// TwinCAT 3 PLC project ConvergeStation
// ProgramVersion: 3.1.4026.26
// libraries:
//   Tc2_ModbusRTU, * (Beckhoff Automation GmbH)
//   Tc2_ModbusSrv, * (Beckhoff Automation GmbH)
//   Tc2_Standard, * (Beckhoff Automation GmbH)
//   Tc2_System, * (Beckhoff Automation GmbH)
// project tree:
//   DUTs/ ST_Outputs.TcDUT
//   GVLs/ GVL.TcGVL, IO.TcGVL
//   / PlcTask.TcTTO
//   POUs/Function Blocks/ FB_Intlk.TcPOU, FB_Motors.TcPOU, FB_Sensors.TcPOU
//   POUs/ MAIN.TcPOU
//   POUs/COMM/ FIO_Read_Inputs.TcPOU, FIO_Write_Outputs.TcPOU, ReadWriteIO.TcPOU
//   POUs/PRG/PRG_CTRL/ PRG_CONTROLM1.TcPOU
//   POUs/PRG/ PRG_Mainprg.TcPOU
//   POUs/PRG/PRG_MOTORS/ PRG_Conveyor01.TcPOU, PRG_ExitConvetor.TcPOU, PRG_Load01.TcPOU, PRG_Conveyor02.TcPOU, PRG_Load02.TcPOU, PRG_TransferLeft02.TcPOU, PRG_TransferLeft01.TcPOU
//   POUs/PRG/PRG_SENSORS/ PRG_AtEntry01.TcPOU, PRG_AtExit01.TcPOU, PRG_AtEntry02.TcPOU, PRG_AtTransfer02.TcPOU, PRG_AtTransfer01.TcPOU
// real-time tasks:
//   TASK PlcTask: cycle T#10ms, priority 20, ADS port 350

CONFIGURATION ConvergeStation
    RESOURCE PLC ON TwinCAT3
        TASK PlcTask(INTERVAL := T#10ms, PRIORITY := 20);
        PROGRAM MAIN WITH PlcTask : MAIN;
    END_RESOURCE
END_CONFIGURATION

// ---- DUTs/ST_Outputs.TcDUT
TYPE ST_Outputs :
STRUCT
	Conveyor_1 : BOOL;
	Load_1 : BOOL;
	Unload_1 : BOOL;
	Transfer_Right_1 : BOOL;
	Transfer_Left_1 : BOOL;
	Conveyor_2: BOOL;
	Load_2 : BOOL;
	Unload_2 : BOOL;
	Transfer_Right_2 : BOOL;
	Transfer_Left_2 : BOOL;
	Exit_Conveyor: BOOL;
	Start_Light: BOOL;
	Reset_Light : BOOL;
	Stop_Light: BOOL;
	Counter : INT;
END_STRUCT
END_TYPE

// ---- GVLs/GVL.TcGVL
{attribute 'qualified_only'}
VAR_GLOBAL
	ReadInputs : FB_MBReadInputs;
	WriteCoils : FB_MBWriteCoils;
	FIO_Inputs : ARRAY [0..15] OF BYTE;
	FIO_Outputs : ARRAY [0..15] OF BYTE;
	StartMachine : BOOL;
	Conveyor01OKToRun : BOOL;
	Conveyor02OKToRun : BOOL;
	AtExitPulse : BOOL;
	TransferOKToStart : BOOL;
END_VAR

// ---- GVLs/IO.TcGVL

VAR_GLOBAL
	At_Entry_1 : BOOL;
	At_Entry_2 : BOOL;
	At_Transfer_1 : BOOL;
	At_Transfer_2 : BOOL;
	At_Exit : BOOL;
	Start : BOOL;
	Reset : BOOL;
	Stop : BOOL;
	Emergency_Stop : BOOL;
	Auto : BOOL;
	
	Conveyor_1 : BOOL;
	Load_1 : BOOL;
	Unload_1 : BOOL;
	Transfer_Right_1 : BOOL;
	Transfer_Left_1 : BOOL;
	Conveyor_2 : BOOL;
	Load_2 : BOOL;
	Unload_2 : BOOL;
	Transfer_Right_2 : BOOL;
	Transfer_Left_2 : BOOL;
	Exit_Conveyor : BOOL;
	Start_Light : BOOL;
	Reset_Light : BOOL;
	Stop_Light : BOOL;
END_VAR

// ---- POUs/MAIN.TcPOU
PROGRAM MAIN
VAR
END_VAR

PRG_Mainprg();
PRG_CONTROLM1();

FIO_Read_Inputs();
FIO_Write_Outputs();
ReadWriteIO();

END_PROGRAM

// ---- POUs/PRG/PRG_Mainprg.TcPOU
PROGRAM PRG_Mainprg
VAR
END_VAR

PRG_Conveyor01();
PRG_Conveyor02();
PRG_ExitConvetor();
PRG_Load01();
PRG_Load02();
PRG_TransferLeft01();
PRG_TransferLeft02();

PRG_AtEntry01();
PRG_AtEntry02();
PRG_AtExit01();
PRG_AtTransfer01();
PRG_AtTransfer02();

END_PROGRAM

// ---- POUs/PRG/PRG_MOTORS/PRG_Conveyor01.TcPOU
PROGRAM PRG_Conveyor01
VAR
	intnFBMotor : FB_Motors;
	intnFBIntlk : FB_Intlk;
END_VAR

intnFBIntlk (
	BackwardsInterlock01 := TRUE,
	BackwardsInterlock02 := TRUE,
	BackwardsInterlock03 := TRUE,
	BackwardsInterlock04 := TRUE,
	BackwardsInterlock05 := TRUE,
	ForwardInterlock01 := GVL.Conveyor01OKToRun,
	ForwardInterlock02 := TRUE,
	ForwardInterlock03 := TRUE,
	ForwardInterlock04 := TRUE,
	ForwardInterlock05 := TRUE,
	oStsInterlockOK => intnFBMotor.inIntlkOK,
);

intnFBMotor (
	inStart := GVL.StartMachine,
	outOTE => Conveyor_1,
);

END_PROGRAM

// ---- POUs/Function Blocks/FB_Motors.TcPOU
FUNCTION_BLOCK FB_Motors
VAR_INPUT
	inIntlkOK : BOOL;
	inStart : BOOL;
END_VAR
VAR_OUTPUT
	outOTE: BOOL;
	outRunning : bool;
	outStopped : BOOL;
END_VAR
VAR
END_VAR

IF inIntlkOK AND inStart THEN
	outOTE := TRUE;
	outRunning := TRUE;
	outStopped := FALSE;
	ELSE
	outStopped := TRUE;
	outRunning := FALSE;
	outOTE := FALSE;
END_IF

END_FUNCTION_BLOCK

// ---- POUs/Function Blocks/FB_Intlk.TcPOU
FUNCTION_BLOCK PUBLIC FB_Intlk
VAR_INPUT
	ForwardInterlock01, ForwardInterlock02, ForwardInterlock03, ForwardInterlock04, ForwardInterlock05: BOOL;
	BackwardsInterlock01, BackwardsInterlock02, BackwardsInterlock03, BackwardsInterlock04, BackwardsInterlock05 : BOOL;
END_VAR
VAR_OUTPUT
	oStsInterlockOK : BOOL;
END_VAR
VAR
END_VAR

oStsInterlockOK := 	ForwardInterlock01 AND 
					ForwardInterlock02 AND 
					ForwardInterlock03 AND 
					ForwardInterlock04 AND 
					ForwardInterlock05 AND 
					BackwardsInterlock01 AND 
					BackwardsInterlock02 AND 
					BackwardsInterlock03 AND 
					BackwardsInterlock04 AND 
					BackwardsInterlock05;

END_FUNCTION_BLOCK

// ---- POUs/PRG/PRG_MOTORS/PRG_Conveyor02.TcPOU
PROGRAM PRG_Conveyor02
VAR
	intnFBMotor : FB_Motors;
	intnFBIntlk : FB_Intlk;
END_VAR

intnFBIntlk (
	BackwardsInterlock01 := TRUE,
	BackwardsInterlock02 := TRUE,
	BackwardsInterlock03 := TRUE,
	BackwardsInterlock04 := TRUE,
	BackwardsInterlock05 := TRUE,
	ForwardInterlock01 := GVL.Conveyor02OKToRun,
	ForwardInterlock02 := TRUE,
	ForwardInterlock03 := TRUE,
	ForwardInterlock04 := TRUE,
	ForwardInterlock05 := TRUE,
	oStsInterlockOK => intnFBMotor.inIntlkOK,
);

intnFBMotor (
	inStart := GVL.StartMachine,
	outOTE => Conveyor_2,
);

END_PROGRAM

// ---- POUs/PRG/PRG_MOTORS/PRG_ExitConvetor.TcPOU
PROGRAM PRG_ExitConvetor
VAR
	intnFBMotor : FB_Motors;
	intnFBIntlk : FB_Intlk;
END_VAR

intnFBIntlk (
	BackwardsInterlock01 := TRUE,
	BackwardsInterlock02 := TRUE,
	BackwardsInterlock03 := TRUE,
	BackwardsInterlock04 := TRUE,
	BackwardsInterlock05 := TRUE,
	ForwardInterlock01 := TRUE,
	ForwardInterlock02 := TRUE,
	ForwardInterlock03 := TRUE,
	ForwardInterlock04 := TRUE,
	ForwardInterlock05 := TRUE,
	oStsInterlockOK => intnFBMotor.inIntlkOK,
);

intnFBMotor (
	inStart := GVL.StartMachine,
	outOTE => Exit_Conveyor,
);

END_PROGRAM

// ---- POUs/PRG/PRG_MOTORS/PRG_Load01.TcPOU
PROGRAM PRG_Load01
VAR
	intnFBMotor : FB_Motors;
	intnFBIntlk : FB_Intlk;
END_VAR

intnFBIntlk (
	BackwardsInterlock01 := TRUE,
	BackwardsInterlock02 := TRUE,
	BackwardsInterlock03 := TRUE,
	BackwardsInterlock04 := TRUE,
	BackwardsInterlock05 := TRUE,
	ForwardInterlock01 := NOT PRG_TransferLeft01.intnFBMotor.outRunning,
	ForwardInterlock02 := TRUE,
	ForwardInterlock03 := TRUE,
	ForwardInterlock04 := TRUE,
	ForwardInterlock05 := TRUE,
	oStsInterlockOK => intnFBMotor.inIntlkOK,
);

intnFBMotor (
	inStart := GVL.StartMachine,
	outOTE => Load_1,
);

END_PROGRAM

// ---- POUs/PRG/PRG_MOTORS/PRG_TransferLeft01.TcPOU
PROGRAM PRG_TransferLeft01
VAR
	intnFBMotor : FB_Motors;
	intnFBIntlk : FB_Intlk;
END_VAR

intnFBIntlk (
	BackwardsInterlock01 := TRUE,
	BackwardsInterlock02 := TRUE,
	BackwardsInterlock03 := TRUE,
	BackwardsInterlock04 := TRUE,
	BackwardsInterlock05 := TRUE,
	ForwardInterlock01 := PRG_TransferLeft02.intnFBMotor.outRunning,
	ForwardInterlock02 := TRUE,
	ForwardInterlock03 := TRUE,
	ForwardInterlock04 := TRUE,
	ForwardInterlock05 := TRUE,
	oStsInterlockOK => intnFBMotor.inIntlkOK,
);

intnFBMotor (
	inStart := GVL.StartMachine,
	outOTE => Transfer_Left_1,
);

END_PROGRAM

// ---- POUs/PRG/PRG_MOTORS/PRG_TransferLeft02.TcPOU
PROGRAM PRG_TransferLeft02
VAR
	intnFBMotor : FB_Motors;
	intnFBIntlk : FB_Intlk;
END_VAR

intnFBIntlk (
	BackwardsInterlock01 := TRUE,
	BackwardsInterlock02 := TRUE,
	BackwardsInterlock03 := TRUE,
	BackwardsInterlock04 := TRUE,
	BackwardsInterlock05 := TRUE,
	ForwardInterlock01 := NOT PRG_AtTransfer01.intnFBSensor.outSensorON OR NOT PRG_AtEntry01.intnFBSensor.outSensorON,
	ForwardInterlock02 := PRG_AtTransfer02.intnFBSensor.outSensorON OR NOT PRG_Load02.intnFBMotor.outRunning,
	ForwardInterlock03 := NOT PRG_AtTransfer01.intnFBSensor.outSensorON AND NOT PRG_AtEntry01.intnFBSensor.outSensorON OR NOT PRG_AtExit01.intnFBSensor.outSensorON,
	ForwardInterlock04 := GVL.TransferOKToStart,
	ForwardInterlock05 := TRUE,
	oStsInterlockOK => intnFBMotor.inIntlkOK,
);

intnFBMotor (
	inStart := GVL.StartMachine AND PRG_AtTransfer02.intnFBSensor.outSensorON OR PRG_TransferLeft01.intnFBMotor.outRunning,
	outOTE => Transfer_Left_2,
);

END_PROGRAM

// ---- POUs/PRG/PRG_SENSORS/PRG_AtTransfer01.TcPOU
PROGRAM PRG_AtTransfer01
VAR
	intnFBSensor : FB_Sensors;
END_VAR

intnFBSensor (
	iSensor := At_Transfer_1,
	iTimeToActuateSensor := 0,
);

END_PROGRAM

// ---- POUs/Function Blocks/FB_Sensors.TcPOU
FUNCTION_BLOCK PUBLIC FB_Sensors
VAR_INPUT
	iSensor : BOOL;
	iTimeToActuateSensor : INT;
END_VAR
VAR_OUTPUT
	outSensorON : BOOL;
END_VAR
VAR
	intnTimer : TON;
END_VAR

intnTImer (
	IN := iSensor,
	PT := INT_TO_TIME(iTimeToActuateSensor),
);

IF iSensor AND intnTimer.Q THEN
	outSensorON := TRUE;
ELSE
	outSensorON := FALSE;	
END_IF

END_FUNCTION_BLOCK

// ---- POUs/PRG/PRG_SENSORS/PRG_AtEntry01.TcPOU
PROGRAM PRG_AtEntry01
VAR
	intnFBSensor : FB_Sensors;
	FEdge : F_TRIG;
	REdge : R_TRIG;
	RTrigPulse : bool;
END_VAR

intnFBSensor (
	iSensor := At_Entry_1,
	iTimeToActuateSensor := 0,
);

FEdge (
	CLK := intnFBSensor.outSensorON,
);

REdge (
	CLK :=  intnFBSensor.outSensorON,
	Q => RTrigPulse,
);

END_PROGRAM

// ---- POUs/PRG/PRG_SENSORS/PRG_AtTransfer02.TcPOU
PROGRAM PRG_AtTransfer02
VAR
	intnFBSensor : FB_Sensors;
END_VAR

intnFBSensor (
	iSensor := At_Transfer_2,
	iTimeToActuateSensor := 0,
);

END_PROGRAM

// ---- POUs/PRG/PRG_MOTORS/PRG_Load02.TcPOU
PROGRAM PRG_Load02
VAR
	intnFBMotor : FB_Motors;
	intnFBIntlk : FB_Intlk;
END_VAR

intnFBIntlk (
	BackwardsInterlock01 := TRUE,
	BackwardsInterlock02 := TRUE,
	BackwardsInterlock03 := TRUE,
	BackwardsInterlock04 := TRUE,
	BackwardsInterlock05 := TRUE,
	ForwardInterlock01 := NOT PRG_AtTransfer02.intnFBSensor.outSensorON,
	ForwardInterlock02 := NOT PRG_TransferLeft02.intnFBMotor.outRunning,
	ForwardInterlock03 := TRUE,
	ForwardInterlock04 := TRUE,
	ForwardInterlock05 := TRUE,
	oStsInterlockOK => intnFBMotor.inIntlkOK,
);

intnFBMotor (
	inStart := GVL.StartMachine,
	outOTE => Load_2,
);

END_PROGRAM

// ---- POUs/PRG/PRG_SENSORS/PRG_AtExit01.TcPOU
PROGRAM PRG_AtExit01
VAR
	intnFBSensor : FB_Sensors;
	FEdge : F_TRIG;
END_VAR

intnFBSensor (
	iSensor := At_Exit,
	iTimeToActuateSensor := 0,
);

FEdge (
	CLK := intnFBSensor.outSensorON,
	Q => GVL.AtExitPulse,
);

END_PROGRAM

// ---- POUs/PRG/PRG_SENSORS/PRG_AtEntry02.TcPOU
PROGRAM PRG_AtEntry02
VAR
	intnFBSensor : FB_Sensors;
	FEdge : F_TRIG;
END_VAR

intnFBSensor (
	iSensor := At_Entry_2,
	iTimeToActuateSensor := 0,
);

FEdge (
	CLK := intnFBSensor.outSensorON,
);

END_PROGRAM

// ---- POUs/PRG/PRG_CTRL/PRG_CONTROLM1.TcPOU
PROGRAM PRG_CONTROLM1
VAR
	TransferStart : TON;
	InTransferStartTimer : BOOL;
	OkTOKeepTransfering : BOOL;
	OkToStartTransfer : BOOL;
END_VAR

IF Auto AND Start THEN
	GVL.StartMachine := TRUE;
END_IF

IF Auto AND NOT Stop OR Reset THEN
	GVL.StartMachine := FALSE;
END_IF

IF GVL.StartMachine THEN
	
	// conveyor 1 ok to start
	IF (PRG_TransferLeft01.intnFBMotor.outRunning AND 
		PRG_TransferLeft02.intnFBMotor.outRunning AND 
			(PRG_AtTransfer01.intnFBSensor.outSensorON OR
 			PRG_AtEntry01.intnFBSensor.outSensorON)) THEN
		
		GVL.Conveyor01OKToRun := FALSE;
		
	ELSIF ((PRG_TransferLeft01.intnFBMotor.outRunning AND 
			PRG_TransferLeft02.intnFBMotor.outRunning) AND 
			(NOT PRG_AtTransfer01.intnFBSensor.outSensorON AND
 			PRG_AtEntry01.intnFBSensor.outSensorON)) THEN
			
		GVL.Conveyor01OKToRun := FALSE;	
		
	ELSIF (PRG_TransferLeft01.intnFBMotor.outRunning AND 
			PRG_TransferLeft02.intnFBMotor.outRunning AND 
			(PRG_AtEntry01.intnFBSensor.outSensorON OR 
			PRG_AtTransfer01.intnFBSensor.outSensorON)) THEN
			
		GVL.Conveyor01OKToRun := FALSE;
		
	ELSE
		
		GVL.Conveyor01OKToRun := TRUE;	
		
	END_IF
	
	// conveyor 2 ok to start	
	IF ((PRG_TransferLeft01.intnFBMotor.outRunning AND 
		PRG_TransferLeft02.intnFBMotor.outRunning) AND 
		PRG_AtEntry02.intnFBSensor.outSensorON) THEN
		
		GVL.Conveyor02OKToRun := FALSE;
		
	ELSIF (PRG_AtTransfer02.intnFBSensor.outSensorON AND 
			PRG_AtEntry02.intnFBSensor.outSensorON) THEN
			
		GVL.Conveyor02OKToRun := FALSE;
		
	ELSE
		
		GVL.Conveyor02OKToRun := TRUE;
		
	END_IF
			
END_IF

// ok to transfer left
IF (PRG_AtExit01.intnFBSensor.outSensorON OR 
	PRG_AtTransfer01.intnFBSensor.outSensorON) AND 
	PRG_ExitConvetor.intnFBMotor.outRunning THEN
	
	GVL.TransferOKToStart := FALSE;
	
ELSIF PRG_AtEntry01.intnFBSensor.outSensorON AND 
	PRG_AtTransfer01.intnFBSensor.outSensorON AND  
	PRG_Conveyor01.intnFBMotor.outRunning THEN
	
	GVL.TransferOKToStart := FALSE;
	
ELSIF (PRG_TransferLeft01.intnFBMotor.outRunning AND 
		PRG_TransferLeft02.intnFBMotor.outRunning AND 
		PRG_AtTransfer01.intnFBSensor.outSensorON) THEN	
		
	GVL.TransferOKToStart := FALSE;
	
ELSIF (NOT PRG_TransferLeft01.intnFBMotor.outRunning AND NOT 
	PRG_TransferLeft02.intnFBMotor.outRunning AND 
	PRG_AtEntry01.intnFBSensor.outSensorON AND 
	PRG_Conveyor01.intnFBMotor.outRunning) THEN
	
	GVL.TransferOKToStart := FALSE;
	
ELSE
	
	GVL.TransferOKToStart := TRUE;	
	
END_IF

END_PROGRAM

// ---- POUs/COMM/FIO_Read_Inputs.TcPOU
PROGRAM FIO_Read_Inputs
VAR
	
	ReadInputsErrorID: UDINT;
END_VAR

GVL.ReadInputs (
	sIPAddr := '127.0.0.1',
	nTCPPort := 505,
	nUnitID := 255,
	nQuantity := 16,
	nMBAddr := 0,
	cbLength := SIZEOF(GVL.FIO_Inputs),
	pDestAddr := ADR(GVL.FIO_Inputs),
	bExecute := TRUE,
	tTimeout := T#1S,
	bBusy => ,
	bError => ,
	nErrId => ReadInputsErrorID,
	cbRead => ,
);
GVL.ReadInputs(bExecute := FALSE);

END_PROGRAM

// ---- POUs/COMM/FIO_Write_Outputs.TcPOU
PROGRAM FIO_Write_Outputs
VAR
	
	WriteCoilsErrorID: UDINT;
END_VAR

GVL.WriteCoils (
	sIPAddr := '127.0.0.1',
	nTCPPort := 505,
	nUnitID := 255,
	nQuantity := 16,
	nMBAddr := 0,
	cbLength := SIZEOF(GVL.FIO_Outputs),
	pSrcAddr := ADR(GVL.FIO_Outputs),
	bExecute := TRUE,
	tTimeout := T#1S,
	bBusy => ,
	bError => ,
	nErrId => WriteCoilsErrorID
	
);
GVL.WriteCoils(bExecute := FALSE);

END_PROGRAM

// ---- POUs/COMM/ReadWriteIO.TcPOU
PROGRAM ReadWriteIO
VAR
END_VAR

//LE AS ENTRADAS
At_Entry_1 := TO_BOOL(GVL.FIO_Inputs[0].0);
At_Entry_2 := TO_BOOL(GVL.FIO_Inputs[0].1);
At_Transfer_1 := TO_BOOL(GVL.FIO_Inputs[0].2);
At_Transfer_2 := TO_BOOL(GVL.FIO_Inputs[0].3);
At_Exit := TO_BOOL(GVL.FIO_Inputs[0].4);
Start := TO_BOOL(GVL.FIO_Inputs[0].5);
Reset := TO_BOOL(GVL.FIO_Inputs[0].6);
Stop := TO_BOOL(GVL.FIO_Inputs[0].7);
Emergency_Stop := TO_BOOL(GVL.FIO_Inputs[1].0);
Auto := TO_BOOL(GVL.FIO_Inputs[1].1);

//LE AS SAÌDAS 
GVL.FIO_Outputs[0].0 := TO_BIT(Conveyor_1);
GVL.FIO_Outputs[0].1 := TO_BIT(Load_1);
GVL.FIO_Outputs[0].2 := TO_BIT(Unload_1);
GVL.FIO_Outputs[0].3 := TO_BIT(Transfer_Right_1);
GVL.FIO_Outputs[0].4 := TO_BIT(Transfer_Left_1);
GVL.FIO_Outputs[0].5 := TO_BIT(Conveyor_2);
GVL.FIO_Outputs[0].6 := TO_BIT(Load_2);
GVL.FIO_Outputs[1].7 := TO_BIT(Unload_2);
GVL.FIO_Outputs[1].0 := TO_BIT(Transfer_Right_2);
GVL.FIO_Outputs[1].1 := TO_BIT(Transfer_Left_2);
GVL.FIO_Outputs[1].2 := TO_BIT(Exit_Conveyor);
GVL.FIO_Outputs[1].3 := TO_BIT(Start_Light);
GVL.FIO_Outputs[1].4 := TO_BIT(Reset_Light);
GVL.FIO_Outputs[1].5 := TO_BIT(Stop_Light);

END_PROGRAM
